INTERFACE I_MotionAxis


METHOD GetPowerOverride : LREAL
END_METHOD

PROPERTY MeasuredAcceleration : LREAL
GET
END_GET
END_PROPERTY

PROPERTY MeasuredPosition : LREAL
GET
END_GET
END_PROPERTY

PROPERTY MeasuredVelocity : LREAL
GET
END_GET
END_PROPERTY


METHOD MoveAbsolute
VAR_INPUT
    Position : LREAL; 
    Velocity : LREAL; 
    Acceleration : LREAL := 0.0; 
    Deceleration : LREAL := 0.0; 
    Jerk : LREAL := 0.0;
    BufferMode : MC_BufferMode := MC_BufferMode.MC_Aborting;
END_VAR
VAR_OUTPUT
    Done : BOOL;
    Busy : BOOL;
    Active : BOOL;
    CommandAborted : BOOL;
    Error : BOOL;
    ErrorID : UDINT;
    ErrorStr : T_MaxString;
END_VAR
END_METHOD

PROPERTY MoveAbsoluteBusy : BOOL
GET
END_GET
END_PROPERTY

PROPERTY MoveAbsoluteDone : BOOL
GET
END_GET
END_PROPERTY

PROPERTY MoveAbsoluteError : BOOL
GET
END_GET
END_PROPERTY

PROPERTY MoveAbsoluteErrorID : UDINT
GET
END_GET
END_PROPERTY

PROPERTY MoveAbsoluteTargetAcceleration : LREAL
GET
END_GET
END_PROPERTY

PROPERTY MoveAbsoluteTargetDeceleration : LREAL
GET
END_GET
END_PROPERTY

PROPERTY MoveAbsoluteTargetJerk : LREAL
GET
END_GET
END_PROPERTY

PROPERTY MoveAbsoluteTargetPosition : LREAL
GET
END_GET
END_PROPERTY

PROPERTY MoveAbsoluteTargetVelocity : LREAL
GET
END_GET
END_PROPERTY

PROPERTY NegativeMotionIsEnabled : BOOL
GET
END_GET
END_PROPERTY

PROPERTY PositiveMotionIsEnabled : BOOL
GET
END_GET
END_PROPERTY


METHOD Power
VAR_INPUT
    Enable : BOOL;
    Enable_Positive : BOOL;
    Enable_Negative : BOOL;
    Override : LREAL := 100.0; (* in percent from 0 to 100 *)
    BufferMode : MC_BufferMode := MC_BufferMode.MC_Aborting;
END_VAR
VAR_OUTPUT
    Status : BOOL;
    Busy : BOOL;
    Active : BOOL;
    Error : BOOL;
    ErrorID : UDINT;
    ErrorStr : T_MaxString;
END_VAR
END_METHOD

PROPERTY PowerError : BOOL
GET
END_GET
END_PROPERTY

PROPERTY PowerErrorID : UDINT
GET
END_GET
END_PROPERTY

PROPERTY PowerIsEnabled : BOOL
GET
END_GET
END_PROPERTY

PROPERTY PowerOverride : LREAL
GET
END_GET
END_PROPERTY

PROPERTY PowerStatus : BOOL
GET
END_GET
END_PROPERTY


METHOD Reset
VAR_OUTPUT
    Done    : BOOL;
    Busy    : BOOL;
    Error   : BOOL;
    ErrorID : UDINT;
    ErrorStr : T_MaxString;
END_VAR
END_METHOD

{warning 'Add property implementation'}
PROPERTY SetpointAcceleration : LREAL
GET
END_GET
END_PROPERTY

{warning 'Add property implementation'}
PROPERTY SetpointJerk : LREAL
GET
END_GET
END_PROPERTY

{warning 'Add property implementation'}
PROPERTY SetpointPosition : LREAL
GET
END_GET
END_PROPERTY

{warning 'Add property implementation'}
PROPERTY SetpointVelocity : LREAL
GET
END_GET
END_PROPERTY


METHOD SetPowerOverride
VAR_INPUT
    Override : LREAL; (* in percent from 0 to 100 *)
END_VAR
VAR_OUTPUT
    Status : BOOL;
    Busy : BOOL;
    Active : BOOL;
    Error : BOOL;
    ErrorID : UDINT;
    ErrorStr : T_MaxString;
END_VAR
END_METHOD

END_INTERFACE

(* stored: Version 1.1.0.1
   Itf I_MotionAxis: Id {4f84f724-7938-4847-ac53-18866323f75e}
   Method GetPowerOverride: Id {d60cf776-350d-4425-919a-ad25cd1e5db1}
   Property MeasuredAcceleration: Id {fb3a018d-3c22-4443-a8e5-6e3745cad979}
   Get Get: Id {eb442b1c-5613-4034-a628-fde5d8279698}
   Property MeasuredPosition: Id {530afb46-d9f4-49ab-80c5-13cb256d3bd1}
   Get Get: Id {15de32b0-7be1-4271-a017-ad85219a0c05}
   Property MeasuredVelocity: Id {e3c7c685-76f5-48ef-a045-ea52f6e128f5}
   Get Get: Id {908664a2-a045-4bc0-be81-065ba84981df}
   Method MoveAbsolute: Id {1eeced1d-efd0-4ca8-90ed-573a0f3007ea}
   Property MoveAbsoluteBusy: Id {f44751a1-7d82-4f25-8f54-5b778d8a0698}
   Get Get: Id {e3f60515-66db-40eb-9c6b-34f9675ffcab}
   Property MoveAbsoluteDone: Id {a0b733c0-9419-4c3c-9610-ac101f8c06ab}
   Get Get: Id {ebba60ae-4e3d-4517-8782-f21b9c51c401}
   Property MoveAbsoluteError: Id {9a5c85d2-7d92-453a-8172-be9ed9715297}
   Get Get: Id {124bf6c1-44fa-4873-9381-da6e3b65a885}
   Property MoveAbsoluteErrorID: Id {338e7459-94f5-4f18-aaac-7e787102062a}
   Get Get: Id {496807ce-16a0-4f8e-a4bb-7ce1b5efd7c7}
   Property MoveAbsoluteTargetAcceleration: Id {2a1afcc8-bb7f-4c80-82cc-6dc1ce5911c2}
   Get Get: Id {212adec5-6179-40e7-bebc-73ce3642b311}
   Property MoveAbsoluteTargetDeceleration: Id {55375e60-2619-4de8-bd6a-d4cedbe4bd56}
   Get Get: Id {ff0bdb1b-e023-4589-a769-b7ce5f0b9853}
   Property MoveAbsoluteTargetJerk: Id {069c0ed3-a231-4195-9a5b-ebca14769a36}
   Get Get: Id {eb6382b4-4294-427e-99d9-b2236c2ea5fb}
   Property MoveAbsoluteTargetPosition: Id {8cc95b48-b223-44d9-8d97-c130c5342454}
   Get Get: Id {ceb3308b-e6ac-49e3-9cd4-2808742b7a81}
   Property MoveAbsoluteTargetVelocity: Id {5951ebaa-5a7a-4a09-99fc-53f37475db1e}
   Get Get: Id {8e1ac7b3-69d1-4497-94cc-dc91b6d2ade0}
   Property NegativeMotionIsEnabled: Id {91b250d2-907a-4479-ae71-ba40251f1e50}
   Get Get: Id {a1c66a4b-626b-4748-87a1-1d44dbd52f26}
   Property PositiveMotionIsEnabled: Id {0491b95b-bf41-4856-b357-395ba3800115}
   Get Get: Id {0c807b83-49c9-486d-adfa-a23a6cc1b724}
   Method Power: Id {b18fd2d7-878f-4d83-b37a-265a5782d415}
   Property PowerError: Id {58e62d80-498f-4d2d-90d8-0787db6c8edd}
   Get Get: Id {15161946-1d82-4920-93f6-7529f20eb627}
   Property PowerErrorID: Id {c7d67a7a-fb66-41ce-8bab-9e318b29d18b}
   Get Get: Id {b5e64e45-9214-49ac-b9d8-6362e9321fb8}
   Property PowerIsEnabled: Id {532451ac-10fb-493a-94cd-9e4135815560}
   Get Get: Id {340aedef-a377-4e4e-a52f-8fdbd3a6026a}
   Property PowerOverride: Id {ed9c07ad-ed08-4877-8e9c-a8fb966768e1}
   Get Get: Id {71360167-1a47-415a-8fb2-8a3280946716}
   Property PowerStatus: Id {5a580bf4-d692-4763-80fe-b7e11f126d99}
   Get Get: Id {aff2e1c1-7432-4f21-8745-b60eb7f95f63}
   Method Reset: Id {16f3e257-dfeb-4005-be51-ff6ea20d250a}
   Property SetpointAcceleration: Id {96d69b8a-074d-4ee2-83da-9ba3d145bc42}
   Get Get: Id {664de77c-602b-4799-9af8-41ed191314bd}
   Property SetpointJerk: Id {52ba8748-9943-4e0f-80ab-781b0227e2d4}
   Get Get: Id {6f4270e7-4109-4b62-936d-01d3124dcb37}
   Property SetpointPosition: Id {5b3af725-cd8d-439c-aea8-05e694f19feb}
   Get Get: Id {1af69962-684c-42ac-977e-e412309c457b}
   Property SetpointVelocity: Id {0aed105f-084d-4362-bfb3-e91c2b94410b}
   Get Get: Id {17353fd9-d464-42ba-af24-dd45833e9d25}
   Method SetPowerOverride: Id {271c429b-7505-4028-9af6-485c3d383120} *)
